{attribute wpf [Container(Layout.Stack)]}
FUNCTION_BLOCK TcoBasicDoor EXTENDS TcoCore.TcoComponent IMPLEMENTS ITcoDoorLock
VAR_IN_OUT
    inoIsClosed : BOOL;
    inoLock : BOOL;
END_VAR
VAR
    {attribute addProperty Name "<#Closed#>"}
    _isClosed : TcoElements.TcoDi(THIS^);

    {attribute addProperty Name "<#Lock#>"}
    _lock : TcoElements.TcoDo(THIS^);


END_VAR

                
THIS^._isClosed(inoSignal :=  inoIsClosed);                    
THIS^._lock(inoSignal   :=  inoLock);

PROPERTY IsClosed : BOOL
GET
IsClosed := THIS^._isClosed.IsTrue;
END_GET
END_PROPERTY

PROPERTY IsLocked : BOOL
GET
IsLocked := THIS^._isClosed.IsTrue and THIS^._lock.IsTrue ;
END_GET
END_PROPERTY

PROPERTY IsOpen : BOOL
GET
IsOpen := THIS^._isClosed.IsFalse;
END_GET
END_PROPERTY

METHOD Lock : BOOL
VAR_INPUT
END_VAR
Lock := FALSE;

THIS^._lock.Set();

IF	THIS^._isClosed.IsTrue THEN 
		Lock := TRUE;
END_IF
END_METHOD

(*~
	<docu>
		<summary>
			Restores this instance to the Ready state. Can be called explicitly or from within one of the restore mechanisms.	
		</summary>			
	</docu>	
~*)
METHOD  Restore : ITcoRestorable
UnLock();
END_METHOD

(*~
	<docu>
		<summary>
		    Custom service (manual, maintenance) logic.
			This method must be implemented in derived class.
		</summary>			
	</docu>	
~*)
METHOD PROTECTED  ServiceMode
END_METHOD

METHOD UnLock : BOOL
VAR_INPUT
END_VAR

UnLock := FALSE;

THIS^._lock.Reset();
		

UnLock := TRUE;
END_METHOD

END_FUNCTION_BLOCK

(* stored: Version 1.1.0.1
   POU TcoBasicDoor: Id {4b9a3f87-7edb-4811-99fe-5791d42a1582}, SpecialFunc None
   Property IsClosed: Id {48ce383b-537a-46e6-bc49-a70d1e2b1ce4}
   Get Get: Id {0f039411-e958-4ce9-85f4-b14d0c5ce179}
   Property IsLocked: Id {c7f6a587-0488-4696-a7ba-8f78ac29c3fc}
   Get Get: Id {b9a2ba96-eac9-48a1-9765-342a91fd2d2b}
   Property IsOpen: Id {7c4462df-1f86-4de1-a3f2-a5d7c8198b38}
   Get Get: Id {fb97a163-d8d6-4766-8b4e-c1569557b630}
   Method Lock: Id {f85d513f-8168-4f0e-ae2a-9722ab75a673}
   Method Restore: Id {f50c15da-9856-42a6-979e-b5230ad38ba2}
   Method ServiceMode: Id {6e28cd51-29d5-449a-8e2b-74f52f0107f1}
   Method UnLock: Id {7b0b1dac-7202-4d6e-b46e-e86ad485d098} *)
